TYPE SignalMapping :
STRUCT
	symbol	: POINTER TO BOOL;
	signal	: POINTER TO Signal;
END_STRUCT
END_TYPE

(* stored: Version 1.1.0.1, ProductVersion 3.1.4024.12
   DUT SignalMapping: Id {4cbc64f9-b243-40a6-93d9-26e2f729a319} *)
